Fanuc KAREL source: CA0110.KL

-- PROVISIONAL review KL for V1013-1; original PC SHA256 021a2e0014adf35423489d5100b05f11d6df4dc504286c80c1b883354c1c974b
-- Incomplete behavior may be omitted. Consult companion uncertainty JSON. Do not deploy.
PROGRAM CA0110
%NOLOCKGROUP
BEGIN
  -- UNRESOLVED_PC offsets 0-1; opcodes 7B
  -- UNRESOLVED_PC offsets 6-16; opcodes 2D,7F
  -- UNRESOLVED_PC offsets 21-25; opcodes 7F
  -- UNRESOLVED_PC offsets 30-37; opcodes 9C,23
  -- UNRESOLVED_PC offsets 42-49; opcodes 9D,23
  -- UNRESOLVED_PC offsets 54-65; opcodes 2E,23
  -- UNRESOLVED_PC offsets 70-77; opcodes 9D,23
  -- UNRESOLVED_PC offsets 82-91; opcodes 3F,75
  -- UNRESOLVED_PC offsets 96-110; opcodes 2E,22,9D,33,35
  -- UNRESOLVED_PC offsets 115-129; opcodes 2E,22,9D,33,35
  -- UNRESOLVED_PC offsets 134-149; opcodes 2E,22,32,35
  -- UNRESOLVED_PC offsets 154-169; opcodes 2E,22,32,35
  -- UNRESOLVED_PC offsets 174-189; opcodes 27,22,AA,79
  -- UNRESOLVED_PC offsets 194-208; opcodes 21,9D,52,23
  -- UNRESOLVED_PC offsets 218-222; opcodes 7F
END CA0110
